FUNCTION_BLOCK FB_TLControl
VAR_INPUT
END_VAR
VAR_OUTPUT
END_VAR
VAR
END_VAR

//Post Startup Logic

IF IO.bEstop_State THEN
	IO_control.bGreenLight := FALSE ;
	IO_control.bYellowLight := FALSE ;
	IO_control.bRedLight := TRUE ;
	IO_control.bBuzzer := TRUE ;
	
ELSIF IO.bInterrupt_State THEN
	IO_control.bGreenLight := FALSE ;
	IO_control.bYellowLight := FALSE ; 
	IO_control.bRedLight := IO.fbBlinker.LightOutput ;
	IO_control.bBuzzer := FALSE ;
	
ELSIF IO_Conveyor.bScan_Failed THEN
	IO_control.bGreenlight := FALSE;
	IO_control.bRedlight := IO.fbBlinker.LightOutput;
	IO_control.bBuzzer := TRUE;
	
ELSIF IO.bAutoMode THEN 
	IO_control.bGreenLight := TRUE ;
	IO_control.bYellowLight := FALSE ;
	IO_control.bRedLight := FALSE ;
	IO_control.bBuzzer := FALSE ;
	
ELSIF IO.bConv_Init_Ready THEN
	IO_control.bGreenLight := FALSE ;
	IO_control.bYellowLight := TRUE ; 
	IO_control.bRedLight := FALSE ;
	IO_control.bBuzzer := FALSE ;

ELSE
	IO_control.bGreenLight := FALSE ;
	IO_control.bYellowLight := TRUE ; 
	IO_control.bRedLight := FALSE ;
	IO_control.bBuzzer := FALSE ;
	
END_IF

END_FUNCTION_BLOCK

(* stored: Version 1.1.0.1, ProductVersion 3.1.4024.12
   POU FB_TLControl: Id {e0ea109f-bc35-4902-98fa-401940ddc42f}, SpecialFunc None *)
